// Reads a bytes field value from the input.
FUNCTION F_WriteBytes : HRESULT
VAR_IN_OUT
    stCtx   : ST_WriteContext;
END_VAR
VAR_IN_OUT CONSTANT    
    aBytes  : ARRAY[*] OF BYTE;
END_VAR
VAR_INPUT
    nLength : UDINT;
END_VAR

F_WriteBytes := S_OK;

F_WriteBytes := F_WriteLength(stCtx, nLength);
IF FAILED(F_WriteBytes) THEN
    RETURN;
END_IF

F_WriteBytes := F_WriteRawBytes(stCtx, F_ToAnyBytes(aBytes), nLength);

END_FUNCTION

(* stored: Version 1.1.0.1
   POU F_WriteBytes: Id {51c66637-48b4-4fb7-bc05-3692f28296d9}, SpecialFunc None *)
